    PROC PlotCirc(num Xcord,num Ycord,num Rad)
        IF ToolNum<>4 THEN
            Home;
            Plotter_Pickup;
        ELSE
            !Check position and move to safe position if needed
            !Check position and move to safe position if needed
            CurrentJoints:=CJointT();
            CurrentPos:=CalcRobT(CurrentJoints,tPlotter\WObj:=Bed1Wyong);

            IF (CurrentPos.trans.z<(Bed1Wyong.uframe.trans.z-30)) OR (((CurrentPos.trans.x+CurrentPos.extax.eax_a)>Bed1Wyong.uframe.trans.x) AND CurrentPos.trans.z<300) THEN
                !Robot in TS
                TPWrite("Jog robot out of tool station AND HOME");
                Stop;
            ENDIF
        ENDIF


        IF Rad<100 THEN
            vPlotter:=[10,5,2000,15];
        ELSE
            vPlotter:=[50,15,2000,15];
        ENDIF


        !Plot Circle
        Plotterc5.trans:=[(-1*Xcord),Ycord,PlotterZ];
        PlotterTemp.trans:=[Plotterc5.trans.x+Rad,Plotterc5.trans.y,PlotterZ];

        IF PlotterTemp.trans.y>0 THEN
            IF PlotterTemp.trans.y<(abs(tPlotter.tframe.trans.x)-10) THEN
                PlotterZOri:=ACos(PlotterTemp.trans.y/abs(tPlotter.tframe.trans.x));
                IF PlotterZOri>PlotA6Max THEN
                    PlotterZOri:=90;
                ENDIF
                PlotterTemp.rot:=OrientZYX(-90+PlotterZOri,0,180);
                PlotterTemp.trans.y:=PlotterTemp.trans.y-((abs(tPlotter.tframe.trans.x)-Ycord)*(9/((abs(tPlotter.tframe.trans.x)-540))));
            ELSEIF PlotterTemp.trans.y<2500 THEN
                PlotterZori:=25;
                PlotterTemp.rot:=OrientZYX(-90+PlotterZOri,0,180);
            ELSE
                PlotterTemp.rot:=OrientZYX(-90,0,180);
            ENDIF
        ELSE
            RAISE ERR_PLOT_POS;
        ENDIF

        IF PlotterTemp.trans.y+Bed1.uframe.trans.y>2800 THEN
            PlotterTemp.extax.eax_a:=(PlotterTemp.trans.x+Bed1Wyong.uframe.trans.x);
        ELSE
            PlotterTemp.extax.eax_a:=(PlotterTemp.trans.x+Bed1Wyong.uframe.trans.x+1000+Abs(tPlotter.tframe.trans.x*Sin(PlotterZOri)));
        ENDIF

        IF PlotterTemp.extax.eax_a>10150 THEN
            PlotterTemp.extax.eax_a:=10100;
        ELSEIF PlotterTemp.extax.eax_a<0 THEN
            PlotterTemp.extax.eax_a:=0;
        ENDIF

        WaitTime\inpos,0.1;
        ConfJ\Off;
        ConfL\Off;

        MoveJ Offs(PlotterTemp,0,0,50),v1500,z5,tPlotter\WObj:=Bed1Wyong;
        MoveL PlotterTemp,v10,fine,tPlotter\WObj:=Bed1Wyong;

        PlotterTemp2.trans:=[Plotterc5.trans.x,Plotterc5.trans.y+Rad,PlotterZ];
        IF PlotterTemp2.trans.y>0 THEN
            IF PlotterTemp2.trans.y<(abs(tPlotter.tframe.trans.x)-10) THEN
                PlotterZOri:=ACos(PlotterTemp2.trans.y/abs(tPlotter.tframe.trans.x));
                IF PlotterZOri>PlotA6Max THEN
                    PlotterZOri:=90;
                ENDIF
                PlotterTemp2.rot:=OrientZYX(-90+PlotterZOri,0,180);
                PlotterTemp2.trans.y:=PlotterTemp2.trans.y-((abs(tPlotter.tframe.trans.x)-(Ycord+Rad))*(9/((abs(tPlotter.tframe.trans.x)-540))));
            ELSEIF PlotterTemp2.trans.y<2500 THEN
                PlotterZori:=25;
                PlotterTemp2.rot:=OrientZYX(-90+PlotterZOri,0,180);
            ELSE
                PlotterZOri:=0;
                PlotterTemp2.rot:=OrientZYX(-90,0,180);
            ENDIF
        ELSE
            RAISE ERR_PLOT_POS;
        ENDIF
        IF PlotterTemp2.trans.y+Bed1.uframe.trans.y>2800 THEN
            PlotterTemp2.extax.eax_a:=(PlotterTemp2.trans.x+Bed1Wyong.uframe.trans.x);
        ELSE
            PlotterTemp2.extax.eax_a:=(PlotterTemp2.trans.x+Bed1Wyong.uframe.trans.x+1000+Abs(tPlotter.tframe.trans.x*Sin(PlotterZOri)));
        ENDIF

        IF PlotterTemp2.extax.eax_a>10150 THEN
            PlotterTemp2.extax.eax_a:=10100;
        ELSEIF PlotterTemp2.extax.eax_a<0 THEN
            PlotterTemp2.extax.eax_a:=0;
        ENDIF

        PlotterTemp3.trans:=[Plotterc5.trans.x-Rad,Plotterc5.trans.y,PlotterZ];
        IF PlotterTemp3.trans.y>0 THEN
            IF PlotterTemp3.trans.y<(abs(tPlotter.tframe.trans.x)-10) THEN
                PlotterZOri:=ACos(PlotterTemp3.trans.y/abs(tPlotter.tframe.trans.x));
                IF PlotterZOri>PlotA6Max THEN
                    PlotterZOri:=90;
                ENDIF
                PlotterTemp3.rot:=OrientZYX(-90+PlotterZOri,0,180);
                PlotterTemp3.trans.y:=PlotterTemp3.trans.y-((abs(tPlotter.tframe.trans.x)-(Ycord-Rad))*(9/((abs(tPlotter.tframe.trans.x)-540))));

            ELSEIF PlotterTemp3.trans.y<2500 THEN
                PlotterZori:=25;
                PlotterTemp3.rot:=OrientZYX(-90+PlotterZOri,0,180);
            ELSE
                PlotterZOri:=0;
                PlotterTemp3.rot:=OrientZYX(-90,0,180);
            ENDIF
        ELSE
            RAISE ERR_PLOT_POS;
        ENDIF
        IF PlotterTemp3.trans.y+Bed1Wyong.uframe.trans.y>2800 THEN
            PlotterTemp3.extax:=[(PlotterTemp3.trans.x+Bed1Wyong.uframe.trans.x),9E+09,9E+09,9E+09,9E+09,9E+09];
        ELSE
            PlotterTemp3.extax:=[(PlotterTemp3.trans.x+Bed1Wyong.uframe.trans.x+1000+Abs(tPlotter.tframe.trans.x*Sin(PlotterZOri))),9E+09,9E+09,9E+09,9E+09,9E+09];
        ENDIF

        IF PlotterTemp3.extax.eax_a>10150 THEN
            PlotterTemp3.extax.eax_a:=10100;
        ELSEIF PlotterTemp3.extax.eax_a<0 THEN
            PlotterTemp3.extax.eax_a:=0;
        ENDIF
        MoveC PlotterTemp2,PlotterTemp3,vPlotter,fine,tPlotter\WObj:=Bed1Wyong;

        PlotterTemp.trans:=[Plotterc5.trans.x,Plotterc5.trans.y-Rad,PlotterZ];
        IF PlotterTemp.trans.y>0 THEN
            IF PlotterTemp.trans.y<(abs(tPlotter.tframe.trans.x)-10) THEN
                PlotterZOri:=ACos(PlotterTemp.trans.y/abs(tPlotter.tframe.trans.x));
                IF PlotterZOri>PlotA6Max THEN
                    PlotterZOri:=90;
                ENDIF
                PlotterTemp.rot:=OrientZYX(-90+PlotterZOri,0,180);
                PlotterTemp.trans.y:=PlotterTemp.trans.y-((abs(tPlotter.tframe.trans.x)-(Ycord-Rad))*(9/((abs(tPlotter.tframe.trans.x)-540))));
            ELSE
                PlotterZOri:=0;
                PlotterTemp.rot:=OrientZYX(-90,0,180);
            ENDIF
        ELSE
            RAISE ERR_PLOT_POS;
        ENDIF

        IF PlotterTemp.trans.y+Bed1.uframe.trans.y>2800 THEN
            PlotterTemp.extax:=[(PlotterTemp.trans.x+Bed1Wyong.uframe.trans.x),9E+09,9E+09,9E+09,9E+09,9E+09];
        ELSE
            PlotterTemp.extax:=[(PlotterTemp.trans.x+Bed1Wyong.uframe.trans.x+1000+Abs(tPlotter.tframe.trans.x*Sin(PlotterZOri))),9E+09,9E+09,9E+09,9E+09,9E+09];
        ENDIF

        IF PlotterTemp.extax.eax_a>10150 THEN
            PlotterTemp.extax.eax_a:=10100;
        ELSEIF PlotterTemp.extax.eax_a<0 THEN
            PlotterTemp.extax.eax_a:=0;
        ENDIF

        PlotterTemp2.trans:=[Plotterc5.trans.x+Rad,Plotterc5.trans.y,PlotterZ];
        IF PlotterTemp2.trans.y>0 THEN
            IF PlotterTemp2.trans.y<(abs(tPlotter.tframe.trans.x)-10) THEN
                PlotterZOri:=ACos(PlotterTemp2.trans.y/abs(tPlotter.tframe.trans.x));
                IF PlotterZOri>PlotA6Max THEN
                    PlotterZOri:=90;
                ENDIF
                PlotterTemp2.rot:=OrientZYX(-90+PlotterZOri,0,180);
                PlotterTemp2.trans.y:=PlotterTemp2.trans.y-((abs(tPlotter.tframe.trans.x)-(Ycord))*(9/((abs(tPlotter.tframe.trans.x)-540))));
            ELSE
                PlotterZOri:=0;
                PlotterTemp2.rot:=OrientZYX(-90,0,180);
            ENDIF
        ELSE
            RAISE ERR_PLOT_POS;
        ENDIF
        IF PlotterTemp2.trans.y+Bed1.uframe.trans.y>2800 THEN
            PlotterTemp2.extax.eax_a:=(PlotterTemp2.trans.x+Bed1Wyong.uframe.trans.x);
        ELSE
            PlotterTemp2.extax.eax_a:=(PlotterTemp2.trans.x+Bed1Wyong.uframe.trans.x+1000+Abs(tPlotter.tframe.trans.x*Sin(PlotterZOri)));
        ENDIF

        IF PlotterTemp2.extax.eax_a>10150 THEN
            PlotterTemp2.extax.eax_a:=10100;
        ELSEIF PlotterTemp2.extax.eax_a<0 THEN
            PlotterTemp2.extax.eax_a:=0;
        ENDIF
        MoveC PlotterTemp,PlotterTemp2,vPlotter,fine,tPlotter\WObj:=Bed1Wyong;
        MoveL Offs(PlotterTemp2,0,0,50),v100,z5,tPlotter\WObj:=Bed1Wyong;
        MoveJ Offs(PlotterTemp2,0,0,200),v500,fine,tPlotter\WObj:=Bed1Wyong;
        ConfJ\On;
        ConfL\On;

    ERROR
        RAISE ;

    ENDPROC

    PROC PackAway()
        !VAR jointtarget jtTarget;
        Home;
        !jtTarget := [[138.31,-55.47,60.29,-0.02,84.30,-2.02], [9416.99,9E+09,9E+09,9E+09,9E+09,9E+09]];
        !MoveAbsJ jtTarget, v500, fine, tTCMaster;
        MoveJ pHomeLoadout,v500,z50,tTCMaster;
    ERROR
        RAISE ;
    ENDPROC


    PROC Home()
        !Move robot to safe position, drop off any tools, close tool boxes

        TEST ToolNum

        CASE 1:
            !TCmaster
            !Check for any tb lids open and robot in tool stations
            !Move to Home
            CurrentJoints:=CJointT();
            CurrentPos:=CalcRobT(CurrentJoints,tTCMaster\WObj:=wobj0);

            IF (CurrentPos.trans.x)>8000 AND (CurrentPos.trans.z<265) THEN
                TPErase;
                TPWrite("Jog robot out of tool station AND HOME");
                Stop;
            ENDIF

        CASE 2:
            !Heli
            CurrentJoints:=CJointT();
            CurrentPos:=CalcRobT(CurrentJoints,tHeli\WObj:=wobj0);

            IF (CurrentPos.trans.x)>8000 AND CurrentPos.trans.z<125 THEN
                TPWrite("Jog robot out of tool station AND HOME");
                Stop;
            ENDIF

            IF CurrentPos.trans.y>(Bed1.uframe.trans.y+3000) THEN
                MoveL Offs(CurrentPos,0,(3000-CurrentPos.trans.y),50),v10,z5,tHeli\WObj:=wobj0;
                MoveJ Offs(CurrentPos,0,(3000-CurrentPos.trans.y),300-CurrentPos.trans.z),v100,z5,tHeli\WObj:=wobj0;
            ENDIF
            Heli_Dropoff;

        CASE 3:
            !VS

            CurrentJoints:=CJointT();
            CurrentPos:=CalcRobT(CurrentJoints,tVS\WObj:=wobj0);


            IF (CurrentPos.trans.x)>8000 AND CurrentPos.trans.z<265 THEN
                TPErase;
                TPWrite("Jog robot out of tool station AND HOME");
                Stop;
            ELSEIF CurrentPos.trans.z<200 THEN
                MoveL Offs(CurrentPos,0,0,(200-CurrentPos.trans.z)),v500,z5,tVS;

            ENDIF


            VS_Dropoff;


        CASE 4:
            !Plotter

            CurrentJoints:=CJointT();
            CurrentPos:=CalcRobT(CurrentJoints,tPlotter\WObj:=wobj0);

            IF CurrentPos.trans.z<270 AND (CurrentPos.trans.x)<8000 THEN
                MoveL Offs(CurrentPos,0,0,(270-CurrentPos.trans.z)),v500,z5,tPlotter;
            ENDIF

            IF (CurrentPos.trans.x)>8000 AND CurrentPos.trans.z<265 THEN
                TPErase;
                TPWrite("Jog robot out of tool station AND HOME");
                Stop;
            ENDIF

            IF CurrentPos.trans.y>(Bed1.uframe.trans.y+3300) THEN
                MoveL Offs(CurrentPos,0,(3300-CurrentPos.trans.y),50),v10,z5,tPlotter\WObj:=wobj0;
                MoveJ Offs(CurrentPos,0,(3300-CurrentPos.trans.y),1000-CurrentPos.trans.z),v100,z5,tPlotter\WObj:=wobj0;
            ENDIF
            Plotter_Dropoff;

        CASE 5:
            CurrentJoints:=CJointT();
            CurrentPos:=CalcRobT(CurrentJoints,tVac\WObj:=wobj0);

            IF (CurrentPos.trans.x)>8000 AND CurrentPos.trans.z<265 THEN
                TPErase;
                TPWrite("Jog robot out of tool station AND HOME");
                Stop;
            ENDIF
            IF CurrentPos.trans.z<200 AND (CurrentPos.trans.x)<8000 THEN
                MoveL Offs(CurrentPos,0,0,(200-CurrentPos.trans.z)),v500,fine,tVac;
            ENDIF
            CurrentJoints:=CJointT();
            CurrentPos:=CalcRobT(CurrentJoints,tVac\WObj:=wobj0);
            IF CurrentPos.trans.y>(Bed1.uframe.trans.y+3000) THEN
                MoveL Offs(CurrentPos,0,(3000-CurrentPos.trans.y),50),v200,z5,tVac\WObj:=wobj0;
                MoveJ Offs(CurrentPos,0,(3000-CurrentPos.trans.y),700-CurrentPos.trans.z),v200,z5,tVac\WObj:=wobj0;
            ENDIF
            Vac_Dropoff;

        CASE 6:
            CurrentJoints:=CJointT();
            CurrentPos:=CalcRobT(CurrentJoints,tPolish\WObj:=wobj0);


            IF (CurrentPos.trans.x)>8000 AND CurrentPos.trans.z<265 THEN
                TPErase;
                TPWrite("Jog robot out of tool station AND HOME");
                Stop;

            ENDIF
            Polish_Dropoff;

        DEFAULT:
            !Unknown
            RAISE ERR_TC_SELECTION;

        ENDTEST

        MoveJ pHome,v500,fine,tTCMaster;

    ERROR
        RAISE ;

    ENDPROC

    FUNC num PointToPointDist(num px,num py,num x1,num y1)
        !Used to check if point is within helicopter blades

        VAR num Dist;

        Dist:=Sqrt((x1-px)*(x1-px)+(y1-py)*(y1-py));
        RETURN Dist;
    ENDFUNC

    FUNC num HighestArray(num count)
        !Used to determine highest height offset
        VAR num j;
        VAR num HighestValue;
        HighestValue:=HeliZArray{1};
        FOR j FROM 1 TO count DO
            IF HeliZArray{j}>HighestValue THEN
                HighestValue:=HeliZArray{j};
            ENDIF
        ENDFOR
        IF PreviousHighest>HighestValue THEN
            PreviousHighest:=HighestValue;
            RETURN PreviousHighest;
        ELSEIF HighestValue<=-30 THEN
            PreviousHighest:=HighestValue;
            RETURN 0;
        ELSE
            PreviousHighest:=HighestValue;
            RETURN HighestValue;
        ENDIF

    ENDFUNC

    PROC HeliZ(num x1,num y1,bool ResetZArray)
        !Determines height offsets for helicopter movements
        VAR num CloseYPos;
        x1:=Abs(x1);
        IF ResetZArray=TRUE THEN
            HeliZArrayCounter:=1;
            FOR i FROM 1 TO DIM(HeliZArray,1) DO
                HeliZArray{i}:=-50;
            ENDFOR
        ENDIF

        FOR i FROM 1 TO 17 DO
            FOR j FROM 1 TO 4 DO
                IF PointToPointDist(x1,y1,BedZpos{j,i,1},BedZpos{j,i,2})<=HeliBladeWidth/2 THEN
                    HeliZArray{HeliZArrayCounter}:=BedZreads{j,i};
                    Incr HeliZArrayCounter;
                ENDIF
            ENDFOR
        ENDFOR

    ENDPROC

    PROC PlotBedGrid(num Xcord1,num Ycord1,num ZOffset)
        !Used by BedGridPlotter for Z datum
        Plotterp1.trans:=[Xcord1,Ycord1,200+ZOffset];
        !+46

        IF Plotterp1.trans.y>0 THEN
            IF Plotterp1.trans.y<(abs(tPlotter.tframe.trans.x)-10) THEN
                PlotterZOri:=ACos(Plotterp1.trans.y/abs(tPlotter.tframe.trans.x));
                IF PlotterZOri>PlotA6Max THEN
                    PlotterZOri:=90;
                ENDIF
                Plotterp1.rot:=OrientZYX(-90+PlotterZOri,0,180);
            ELSE
                PlotterZOri:=0;
                Plotterp1.rot:=OrientZYX(-90,0,180);
            ENDIF
        ELSE
            RAISE ERR_PLOT_POS;
        ENDIF

        IF PlotterP1.trans.y>(abs(tPlotter.tframe.trans.x)+250) THEN
            Plotterp1.extax:=[(Plotterp1.trans.x+Bed1.uframe.trans.x),9E+09,9E+09,9E+09,9E+09,9E+09];
        ELSE
            Plotterp1.extax:=[(Plotterp1.trans.x+Bed1.uframe.trans.x+1000+Abs(tPlotter.tframe.trans.x*Sin(PlotterZOri))),9E+09,9E+09,9E+09,9E+09,9E+09];
        ENDIF

        IF Plotterp1.extax.eax_a>10150 THEN
            Plotterp1.extax.eax_a:=10100;
        ENDIF

        IF Plotterp1.extax.eax_a<0 THEN
            Plotterp1.extax.eax_a:=0;
        ENDIF

        vPlotter:=[100,15,2000,15];

        MoveL Plotterp1,v300,zPlotter,tTCMaster\WObj:=Bed1Wyong;

    ENDPROC

    PROC BedGridPlotter()
        !Get Z datum offset
        FOR k FROM 7 TO 19 DO
            !Move x
            FOR j FROM 4 TO 9 DO
                !Move y

                PlotBedGrid(k*XGridSpacing+100),(j*YGridSpacing+100),Bed1Zread{10-j,(k+1)};
                WaitTime\inpos,0.1;

            ENDFOR

        ENDFOR

    ENDPROC

    PROC MoveGridDatum()
        !Sweep across bed maintaining Z height through offsets
        FOR j FROM 9 TO 4 DO
            FOR k FROM 11 TO 1 DO
                !Move x
                PlotBedGrid(k*XGridSpacing+100),(j*YGridSpacing+100),Bed1Zread{10-j,(k+1)};
            ENDFOR
        ENDFOR
    ENDPROC


    PROC VacuumBed()

        VAR num VacOverlap:=-400;
        IF ToolNum<>5 THEN
            Home;
            Vac_Pickup;
        ELSE
            CurrentJoints:=CJointT();
            CurrentPos:=CalcRobT(CurrentJoints,tVac\WObj:=Bed1Wyong);
            IF CurrentPos.trans.x<0 AND (CurrentPos.trans.z<150) THEN
                MoveL Offs(CurrentPos,0,0,(150-CurrentPos.trans.z)),v500,z5,tVac\WObj:=Bed1Wyong;
            ELSEIF (CurrentPos.trans.z<700) THEN
                MoveL Offs(CurrentPos,0,0,(700-CurrentPos.trans.z)),v500,z5,tVac\WObj:=Bed1Wyong;
            ENDIF
        ENDIF

        pTemp:=pVacStart;
        pTemp2:=pVacStart;
        pTemp2.trans.x:=pVacStart2.trans.x;
        pTemp2.extax.eax_a:=pVacStart2.extax.eax_a;

        Vac_on;
        FOR i FROM 0 TO (Round((pVacStart.trans.y-pVacStart2.trans.y)/(-1*VacOverlap))) DO
            IF pTemp.trans.y+i*VacOverlap>pVacStart2.trans.y THEN
                MoveJ Offs(pTemp,0,i*VacOverlap,150),v500,z5,tVac\WObj:=Bed1Wyong;
                MoveL Offs(pTemp,0,i*VacOverlap,0),v50,z5,tVac\WObj:=Bed1Wyong;
                MoveL Offs(pTemp2,0,i*VacOverlap,0),v100,z5,tVac\WObj:=Bed1Wyong;
                MoveL Offs(pTemp2,0,i*VacOverlap,150),v50,fine,tVac\WObj:=Bed1Wyong;
            ENDIF
        ENDFOR

        Vac_off;

        CurrentJoints:=CJointT();
        CurrentPos:=CalcRobT(CurrentJoints,tVac\WObj:=wobj0);
        MoveL Offs(CurrentPos,0,0,800-CurrentPos.trans.z),v100,z5,tVac\WObj:=wobj0;

    ENDPROC

    PROC JointPositions()

        VAR num PolishOverlap:=450;
        pPolTemp:=pPolStart1;
        pPolTemp2:=pPolStart1;
        pPolTemp2.extax.eax_a:=pPolStart1.extax.eax_a-7500;
        pPolTemp2.trans.x:=-7500;

        pPolTemp.rot:=pPolStart1.rot;
        pPolTemp2.rot:=pPolStart1.rot;

        pPolTemp2.rot:=pPolStart2.rot;
        pPolTemp2.extax.eax_a:=pPolStart1.extax.eax_a-8500;
        CurrentJoints5:=CJointT();
        CurrentJoints6:=CalcJointT(Offs(pPolTemp2,50,(1+1)*PolishOverlap,40),tPolish\WObj:=Bed1Wyong);

    ENDPROC


    PROC RobbiePlot()

        ! !Write R
        !PlotLine 6900,1000, 6900,2000;
        !PlotArc 6900,2000,6650,1750,6900,1500;
        !PlotLine 6900,1500,6650,1000;

        !!Write O
        !PlotArc 6300,2000, 6050,1500,6300,1000;
        !PlotArc 6300,1000, 6550,1500,6300,2000;

        !!Write B
        !PlotLine 5700,1000, 5700,2000;
        !PlotArc 5700,2000,5450,1750,5700,1500;
        !PlotArc 5700,1500,5450,1250,5700,1000;

        !!Write B
        !PlotLine 5100,1000, 5100,2000;
        !PlotArc 5100,2000,4850,1750,5100,1500;
        !PlotArc 5100,1500,4850,1250,5100,1000;

        !!Write I
        !PlotLine 4500,1000, 4500,2000;

        !!Write E
        !PlotLine 3900,1000, 3900,2000;
        !PlotLine 3900,2000, 3400,2000;
        !PlotLine 3900,1500, 3400,1500;
        !PlotLine 3900,1000, 3400,1000;

        !formbox
        PlotRect 2000,500,2000,3500,6000,3500,6000,500;
        !Ferrule
        WaitTime\inpos,0.1;
        PlotCirc 2250,750,(PlotCircleD/2);
        PlotLine(2250-PlotCircleD/2-CrossHairExt),750,(2250+PlotCircleD/2+CrossHairExt),750;
        PlotLine 2250,(750-PlotCircleD/2-CrossHairExt),2250,(750+PlotCircleD/2+CrossHairExt);
        !Ferrule
        WaitTime\inpos,0.1;
        PlotCirc 2250,3250,(PlotCircleD/2);
        PlotLine(2250-PlotCircleD/2-CrossHairExt),3250,(2250+PlotCircleD/2+CrossHairExt),3250;
        PlotLine 2250,(3250-PlotCircleD/2-CrossHairExt),2250,(3250+PlotCircleD/2+CrossHairExt);
        !Grout tube Casee 4
        WaitTime\inpos,0.1;
        iCoord1x:=6000;
        iCoord1y:=2000;
        iAngle:=0;
        PlotRect iCoord1x-GroutWidth/2*Sin(iAngle)-GroutHeight*Cos(iAngle),iCoord1y+GroutHeight*Sin(iAngle)-GroutWidth/2*Cos(iAngle),iCoord1x+GroutWidth/2*Sin(iAngle)-GroutHeight*Cos(iAngle),iCoord1y+GroutHeight*Sin(iAngle)+GroutWidth/2*Cos(iAngle),iCoord1x+GroutWidth/2*Sin(iAngle),iCoord1y+GroutWidth/2*Cos(iAngle),iCoord1x-GroutWidth/2*Sin(iAngle),iCoord1y-GroutWidth/2*Cos(iAngle);

        !Lifting points 180 angle
        WaitTime\inpos,0.1;
        TriangleAngle:=180;
        iCoord1x:=5000;
        iCoord1y:=3500;
        PlotLine iCoord1x-TriangleHeight*Sin(TriangleAngle),iCoord1y-TriangleHeight*Cos(TriangleAngle),iCoord1x-TriangleBase/2*Cos(TriangleAngle),iCoord1y+TriangleBase/2*Sin(TriangleAngle);
        PlotLine iCoord1x-TriangleBase/2*Cos(TriangleAngle),iCoord1y+TriangleBase/2*Sin(TriangleAngle),iCoord1x+TriangleBase/2*Cos(TriangleAngle),iCoord1y-TriangleBase/2*Sin(TriangleAngle);
        PlotLine iCoord1x+TriangleBase/2*Cos(TriangleAngle),iCoord1y-TriangleBase/2*Sin(TriangleAngle),iCoord1x-TriangleHeight*Sin(TriangleAngle),iCoord1y-TriangleHeight*Cos(TriangleAngle);
        !Lifting points 180 angle
        WaitTime\inpos,0.1;
        TriangleAngle:=180;
        iCoord1x:=3000;
        iCoord1y:=3500;
        PlotLine iCoord1x-TriangleHeight*Sin(TriangleAngle),iCoord1y-TriangleHeight*Cos(TriangleAngle),iCoord1x-TriangleBase/2*Cos(TriangleAngle),iCoord1y+TriangleBase/2*Sin(TriangleAngle);
        PlotLine iCoord1x-TriangleBase/2*Cos(TriangleAngle),iCoord1y+TriangleBase/2*Sin(TriangleAngle),iCoord1x+TriangleBase/2*Cos(TriangleAngle),iCoord1y-TriangleBase/2*Sin(TriangleAngle);
        PlotLine iCoord1x+TriangleBase/2*Cos(TriangleAngle),iCoord1y-TriangleBase/2*Sin(TriangleAngle),iCoord1x-TriangleHeight*Sin(TriangleAngle),iCoord1y-TriangleHeight*Cos(TriangleAngle);

        Plotter_Dropoff;

    ENDPROC

    PROC PolishDemo()
        IF ToolNum<>6 THEN
            Home;
            Polish_Pickup;
        ELSE
            CurrentJoints:=CJointT();
            CurrentPos:=CalcRobT(CurrentJoints,tPolish\WObj:=wobj0);
            IF CurrentPos.trans.z<600 THEN
                MoveL Offs(CurrentPos,0,0,(600-CurrentPos.trans.z)),v500,z5,tPolish;
            ENDIF
        ENDIF
        MoveJ pPolHome,v500,z5,tPolish;
        pPolTemp:=pPolStart1;
        pPolTemp2:=pPolStart1;
        pPolTemp2.extax.eax_a:=pPolStart1.extax.eax_a-7500;
        pPolTemp2.trans.x:=-7500;
        pPolTemp.rot:=pPolStart1.rot;
        pPolTemp2.rot:=pPolStart1.rot;
        FCCalib PolishLoad;
        pPolTemp.extax.eax_a:=pPolStart1.extax.eax_a;
        MoveJ Offs(pPolTemp,0,0,100),v500,z5,tPolish\WObj:=Bed1Wyong;
        Pol_on;
        MoveL Offs(pPolTemp,0,0,50),v100,fine,tPolish\WObj:=Bed1Wyong;
        myForceVector:=FCGetForce(\Tool:=tPolish);
        FCPress1LStart Offs(pPolTemp,-25,0,55),v10,\Fz:=120,15,\ForceChange:=50\PosSupvDist:=125,z5,tPolish\WObj:=Bed1Wyong;
        pPolTemp2.extax.eax_a:=pPolStart2.extax.eax_a-300;
        FCPressL Offs(pPolTemp2,-300,0,-15),v100,130,fine,tPolish\WObj:=Bed1Wyong;
        FCPressEnd Offs(pPolTemp2,-300,0,75),v50,\DeactOnly,tPolish\WObj:=Bed1Wyong;
        CurrentJoints:=CJointT();
        CurrentPos:=CalcRobT(CurrentJoints,tPolish\WObj:=Bed1Wyong);
        MoveJ Offs(Reltool(CurrentPos,0,0,-100),0,450,0),v100,fine,tPolish\WObj:=Bed1Wyong;
        Pol_off;
        Polish_Dropoff;
    ENDPROC



    PROC BedGrid()

        !        MoveJ Offs(p10Maps,500*(1-1)+2000*(1-1),650*(1-1),50),v500,z5,tTCMaster\WObj:=Bed1Wyong;
        !        MoveL Offs(p10Maps,500*(1-1)+2000*(1-1),650*(1-1),0),v500,fine,tTCMaster\WObj:=Bed1Wyong;
        !        Stop;
        !        MoveL Offs(p10Maps,500*(1-1)+2000*(1-1),650*(1-1),50),v500,z5,tTCMaster\WObj:=Bed1Wyong;
        !        Stop;

        FOR i FROM 1 TO 5 DO
            !Move EAX
            FOR k FROM 1 TO 4 DO
                !Move x
                FOR j FROM 1 TO 4 DO
                    !Move y
                    IF 500*(k-1)+2000*(i-1)<8001 THEN
                        p10maps.extax.eax_a:=Bed1Wyong.uframe.trans.x+p10Maps.trans.x-500*(k-1)-2000*(i-1);
                        IF p10maps.extax.eax_a>10150 THEN
                            p10maps.extax.eax_a:=10100;
                        ENDIF
                        IF p10maps.extax.eax_a<1000 THEN
                            p10maps.extax.eax_a:=1000;
                        ENDIF

                        !MoveJ Offs(p10Maps,-500*(k-1)-2000*(i-1),650*(j-1),50),v500,z5,tTCMaster\WObj:=Bed1Wyong;
                        !MoveL Offs(p10Maps,-500*(k-1)-2000*(i-1),650*(j-1),0),v500,fine,tTCMaster\WObj:=Bed1Wyong;
                        !TPReadNum BedZread,"Enter Z reading";
                        !BedZreads{5-j,((i-1)*4+k)}:=BedZread;
                        BedZpos{5-j,((i-1)*4+k),1}:=p10Maps.trans.x-500*(k-1)-2000*(i-1);
                        BedZpos{5-j,((i-1)*4+k),2}:=p10maps.trans.y+650*(j-1);
                        !MoveL Offs(p10Maps,-500*(k-1)-2000*(i-1),650*(j-1),50),v500,z5,tTCMaster\WObj:=Bed1Wyong;
                    ENDIF

                ENDFOR
            ENDFOR
        ENDFOR
        Stop;

    ENDPROC


    PROC ClearBedZ()

        FOR i FROM 1 TO 4 DO
            !Move EAX
            FOR k FROM 1 TO 24 DO
                !Move x
                BedZreads{i,k}:=0;
                BedZpos{i,k,1}:=0;
                BedZpos{i,k,2}:=0;
            ENDFOR
        ENDFOR

    ENDPROC




    PROC BHTestTask()
        TPErase;
        TPWrite "BH Test Task";
        TPWrite "Press Play to confirm and start task";
        Stop;

        TPErase;
        TPWrite "Starting BH Test Task...";

        Heli_Pickup;
        MoveJ Offs(ptHeli,0,0,1000),v500,fine,tHeli;
        TPWrite "Helicopter tool at 1000mm above pickup";
        WaitTime 2;

        Heli_Dropoff;
        TPWrite "Helicopter tool dropped off";

        Polish_Pickup;
        MoveJ Offs(ptPolish,0,0,1000),v500,fine,tPolish;
        TPWrite "Polisher tool at 1000mm above pickup";
        WaitTime 2;

        Polish_Dropoff;
        TPWrite "Polisher tool dropped off";

        Home;
        TPWrite "BH Test Task Complete";

    ERROR
        RAISE ;
    ENDPROC



    PROC Datum()
        ! Datum - draws small circle at Bed1Wyong origin (0,0)
        ! Generated by Onyx Toolpath Generator
        VAR robtarget pDatumCenter;
        VAR robtarget pDatumCircle;
        VAR num DatumZ:=0;
        VAR num DatumRadius:=100;
        VAR num SafeZ:=500;
        VAR num i;

        TPWrite "Datum: ToolNum=" \Num:=ToolNum;
        IF ToolNum<>4 THEN
            TPWrite "No plotter! Will pickup plotter.";
            Stop;
            Home;
            Plotter_Pickup;
        ELSE
            CurrentJoints:=CJointT();
            CurrentPos:=CalcRobT(CurrentJoints,tPlotter\WObj:=wobj0);
            IF CurrentPos.trans.z<600 THEN
                MoveL Offs(CurrentPos,0,0,(600-CurrentPos.trans.z)),v500,z5,tPlotter;
            ENDIF
        ENDIF

        ConfL\Off;
        ConfJ\Off;

        pDatumCenter:=[[0,0,DatumZ],[0,0,1,0],[0,0,0,0],[0,9E+09,9E+09,9E+09,9E+09,9E+09]];
        pDatumCenter.rot:=OrientZYX(-90,0,180);
        pDatumCenter.extax.eax_a:=6500;

        TPWrite "Datum: Drawing circle at origin";
        TPWrite "Press Play to continue";
        Stop;

        pDatumCircle:=pDatumCenter;
        pDatumCircle.trans.z:=SafeZ;
        MoveJ pDatumCircle,v500,z5,tPlotter\WObj:=Bed1Wyong;

        pDatumCircle.trans.x:=DatumRadius;
        pDatumCircle.trans.z:=DatumZ;
        MoveJ pDatumCircle,v500,z5,tPlotter\WObj:=Bed1Wyong;

        FOR i FROM 1 TO 8 DO
            pDatumCircle.trans.x:=DatumRadius*Cos(i*45);
            pDatumCircle.trans.y:=DatumRadius*Sin(i*45);
            MoveJ pDatumCircle,v100,fine,tPlotter\WObj:=Bed1Wyong;
        ENDFOR

        pDatumCircle.trans.x:=0;
        pDatumCircle.trans.y:=0;
        pDatumCircle.trans.z:=DatumZ;
        MoveJ pDatumCircle,v100,fine,tPlotter\WObj:=Bed1Wyong;

        TPWrite "Plotter at datum center (0,0)";
        TPWrite "Press Play to return tool";
        Stop;

        pDatumCircle.trans.z:=SafeZ;
        MoveJ pDatumCircle,v500,z5,tPlotter\WObj:=Bed1Wyong;

        ConfL\On;
        ConfJ\On;

        Plotter_Dropoff;
        Home;

        TPWrite "Datum Complete";
    ERROR
        RAISE;
    ENDPROC


    PROC PyHeli()
        ! PyHeli - Helicopter serpentine pattern
        ! Workzone: panel
        ! Force Control ENABLED: 300N (ramping 10%->100% over 5s)
        ! Generated by Onyx Toolpath Generator

        VAR robtarget pHeliPos;
        VAR robtarget pHeliEnd;
        VAR num HeliZ:=150;
        VAR num SafeZ:=500;

        ! Workspace bounds (with offsets applied)
        VAR num WorkMinX:=1900;
        VAR num WorkMaxX:=6550;
        VAR num WorkMinY:=700;
        VAR num WorkMaxY:=2100;

        ! Pattern parameters
        VAR num StepSize:=450;
        VAR num SweepDir:=1;
        VAR num StepDir:=-1;
        VAR num CurrentY:=2100;
        VAR num CurrentX:=1900;
        VAR num NextY;
        VAR num NextX;
        VAR num StartX;
        VAR num EndX;
        VAR num StartY;
        VAR num EndY;

        ! Speed and blade parameters
        VAR num HeliSpeed:=100;
        VAR num HeliAngle:=8;
        VAR speeddata vHeliTravel:=[500,15,2000,15];
        VAR num NumPasses;
        VAR num HeliForce:=300;
        VAR num CurrentForce:=300;
        VAR clock RampClock;
        VAR bool bRamping:=FALSE;

        NumPasses:=Trunc(Abs(WorkMaxY-WorkMinY)/StepSize)+1;

        TPWrite "PyHeli: Serpentine Pattern";
        TPWrite "Work Area (6550,2100) to (1900,700)";
        TPWrite "Passes=" \Num:=NumPasses;
        TPWrite "Step=" \Num:=StepSize;
        TPWrite "Force=ON 300N";

        IF ToolNum<>2 THEN
            TPWrite "PyHeli: ToolNum<>2, need pickup";
            Stop;
            Home;
            Heli_Pickup;
        ELSE
            CurrentJoints:=CJointT();
            CurrentPos:=CalcRobT(CurrentJoints,tHeli\WObj:=Bed1Wyong);
            IF CurrentPos.trans.z<SafeZ THEN
                MoveL Offs(CurrentPos,0,0,(SafeZ-CurrentPos.trans.z)),v500,z5,tHeli\WObj:=Bed1Wyong;
            ENDIF
        ENDIF

        ! Set start/end based on sweep direction
        IF SweepDir=1 THEN
            StartX:=WorkMinX;
            EndX:=WorkMaxX;
        ELSE
            StartX:=WorkMaxX;
            EndX:=WorkMinX;
        ENDIF

        ! Set initial position with fixed orientation
        pHeliPos:=[[0,0,HeliZ],OrientZYX(0,0,180),[0,0,0,0],[0,9E+09,9E+09,9E+09,9E+09,9E+09]];

        ! Move to row start above surface (HOVER)
        pHeliPos.trans.x:=-StartX;
        pHeliPos.trans.y:=CurrentY;
        pHeliPos.trans.z:=SafeZ;
        pHeliPos.extax.eax_a:=Bed1Wyong.uframe.trans.x-StartX;
        MoveJ pHeliPos,v500,z5,tHeli\WObj:=Bed1Wyong;

        ! Disable configuration tracking for serpentine movements
        ConfL\Off;
        ConfJ\Off;

        ! Home stepper before setting blade angle (ensures StepperPos is valid)
        TPWrite "Homing blade stepper...";
        Heli_Stepper_Home;
        TPWrite "Stepper homed";

        ! Set blade angle while hovering
        TPWrite "Setting blade angle to " \Num:=HeliAngle;
        HeliBlade_Angle HeliAngle;
        WaitTime 2;
        TPWrite "Blade angle set";

        ! Calibrate force sensor while stationary (before blade spin)
        TPWrite "Calibrating force sensor...";
        FCCalib HeliLoad140rpm;
        TPWrite "Force sensor calibrated";

        TPWrite "Hovering over workspace - Press Play to start";
        Stop;

        ! Start blade rotation BEFORE lowering
        TPWrite "Starting blade rotation...";
        HeliBladeSpeed HeliSpeed,"FWD";
        WaitTime 1;

        ! Lower to working height
        TPWrite "Lowering to work surface...";
        pHeliPos.trans.z:=HeliZ;
        MoveL pHeliPos,v50,fine,tHeli\WObj:=Bed1Wyong;

        ! Start force control at 10% of target
        CurrentForce:=HeliForce*0.1;
        FCPress1LStart Offs(pHeliPos,0,0,25),v50,\Fz:=CurrentForce,15,\ForceChange:=50\PosSupvDist:=100,z5,tHeli\WObj:=Bed1Wyong;

        ! Start ramp timer - will ramp to 100% over 5 seconds during first sweep
        ClkReset RampClock;
        ClkStart RampClock;
        bRamping:=TRUE;
        TPWrite "Force ramping: 10% -> 100% over 5s";

        ! Set up end position for first sweep
        pHeliEnd:=pHeliPos;
        pHeliEnd.trans.x:=-EndX;
        pHeliEnd.extax.eax_a:=Bed1Wyong.uframe.trans.x-EndX;

        ! ========== PASS 1: X-direction sweeps (stepping in Y) ===========
        WHILE TRUE DO
            ! === SWEEP X (full length) ===
            FCPressL pHeliEnd,vHeliTravel,CurrentForce,fine,tHeli\WObj:=Bed1Wyong;

            ! Update force ramp if still ramping (applied on next move)
            IF bRamping THEN
                IF ClkRead(RampClock)>=5 THEN
                    CurrentForce:=HeliForce;
                    bRamping:=FALSE;
                    TPWrite "Force ramp complete: " \Num:=CurrentForce;
                ELSE
                    CurrentForce:=HeliForce*(0.1+0.9*ClkRead(RampClock)/5);
                ENDIF
            ENDIF

            ! Calculate next row
            NextY:=CurrentY+(StepDir*StepSize);

            ! Check if pass complete
            IF (StepDir=1 AND NextY>WorkMaxY) OR (StepDir=-1 AND NextY<WorkMinY) THEN
                EXIT;
            ENDIF

            ! Clamp to bounds
            IF NextY>WorkMaxY THEN
                NextY:=WorkMaxY;
            ELSEIF NextY<WorkMinY THEN
                NextY:=WorkMinY;
            ENDIF

            ! Step to next Y row
            pHeliEnd.trans.y:=NextY;
            FCPressL pHeliEnd,vHeliTravel,CurrentForce,fine,tHeli\WObj:=Bed1Wyong;
            CurrentY:=NextY;

            ! Flip sweep direction
            SweepDir:=-SweepDir;
            IF SweepDir=1 THEN
                StartX:=WorkMinX;
                EndX:=WorkMaxX;
            ELSE
                StartX:=WorkMaxX;
                EndX:=WorkMinX;
            ENDIF

            ! Set up end position for next sweep
            pHeliEnd.trans.x:=-EndX;
            pHeliEnd.extax.eax_a:=Bed1Wyong.uframe.trans.x-EndX;
        ENDWHILE

        ! ========== PASS 2: Y-direction sweeps (stepping in X) ==========
        TPWrite "=== PASS 2 START ===";

        ! Reset for Y-direction passes - start from current position
        CurrentX:=Abs(pHeliEnd.trans.x);
        TPWrite "Pass2: CurrentX=" \Num:=CurrentX;
        TPWrite "Pass2: CurrentY=" \Num:=CurrentY;
        TPWrite "Pass2: WorkMinX=" \Num:=WorkMinX;
        TPWrite "Pass2: WorkMaxX=" \Num:=WorkMaxX;

        ! Determine step direction based on where Pass 1 ended
        ! At high X, step toward low X; at low X, step toward high X
        IF CurrentX>((WorkMinX+WorkMaxX)/2) THEN
            StepDir:=-1;
            TPWrite "Pass2: StepDir=-1 (toward MinX)";
        ELSE
            StepDir:=1;
            TPWrite "Pass2: StepDir=+1 (toward MaxX)";
        ENDIF

        ! Determine sweep direction based on where Pass 1 ended (which Y edge)
        IF CurrentY>((WorkMinY+WorkMaxY)/2) THEN
            SweepDir:=1;
            StartY:=WorkMaxY;
            EndY:=WorkMinY;
            TPWrite "Pass2: Sweep MinY first";
        ELSE
            SweepDir:=-1;
            StartY:=WorkMinY;
            EndY:=WorkMaxY;
            TPWrite "Pass2: Sweep MaxY first";
        ENDIF

        TPWrite "Pass2: EndY=" \Num:=EndY;

        ! First Y sweep from current position
        TPWrite "Pass2: First Y sweep...";
        pHeliEnd.trans.y:=EndY;
        FCPressL pHeliEnd,vHeliTravel,CurrentForce,fine,tHeli\WObj:=Bed1Wyong;
        TPWrite "Pass2: First Y sweep done";

        TPWrite "Pass2: Entering X-step loop";

        WHILE TRUE DO
            ! Calculate next column
            NextX:=CurrentX+(StepDir*StepSize);
            TPWrite "Pass2: NextX=" \Num:=NextX;

            ! Check if pass complete (no more columns to step to)
            IF (StepDir=1 AND NextX>WorkMaxX) OR (StepDir=-1 AND NextX<WorkMinX) THEN
                TPWrite "Pass2: EXIT - NextX out of bounds";
                FCPressEnd Offs(pHeliEnd,0,0,50),v100,\DeactOnly,tHeli\WObj:=Bed1Wyong;
                EXIT;
            ENDIF

            ! Clamp to bounds
            IF NextX>WorkMaxX THEN
                NextX:=WorkMaxX;
            ELSEIF NextX<WorkMinX THEN
                NextX:=WorkMinX;
            ENDIF

            ! Step to next X column
            TPWrite "Pass2: Step to X=" \Num:=NextX;
            pHeliEnd.trans.x:=-NextX;
            pHeliEnd.extax.eax_a:=Bed1Wyong.uframe.trans.x-NextX;
            FCPressL pHeliEnd,vHeliTravel,CurrentForce,fine,tHeli\WObj:=Bed1Wyong;
            CurrentX:=NextX;

            ! Flip sweep direction for next Y sweep
            SweepDir:=-SweepDir;
            IF SweepDir=1 THEN
                EndY:=WorkMinY;
            ELSE
                EndY:=WorkMaxY;
            ENDIF

            ! Set up end position and sweep Y
            TPWrite "Pass2: Sweep Y to " \Num:=EndY;
            pHeliEnd.trans.y:=EndY;
            FCPressL pHeliEnd,vHeliTravel,CurrentForce,fine,tHeli\WObj:=Bed1Wyong;
        ENDWHILE
        TPWrite "=== PASS 2 COMPLETE ===";

        ! === LIFT OFF BED ===
        pHeliPos.trans.z:=SafeZ;
        MoveL pHeliPos,v100,z5,tHeli\WObj:=Bed1Wyong;

        ! === STOP BLADE ROTATION ===
        HeliBladeSpeed 0,"FWD";
        WaitTime\InPos,3;

        ConfL\On;
        ConfJ\On;

        ! === PACKAWAY ===
        Heli_Dropoff;
        Home;

        TPWrite "PyHeli Complete";
    ERROR
        HeliBladeSpeed 0,"FWD";
        RAISE;
    ENDPROC


    PROC PyVac()
        ! PyVac - Vacuum procedure with serpentine pattern
        ! Workzone: bed
        ! Generated by Onyx Toolpath Generator

        VAR robtarget pVacPos;
        VAR robtarget pVacEnd;
        VAR num VacZ:=-20;
        VAR num SafeZ:=300;

        ! Force control parameters
        VAR num VacForce:=50;
        VAR num VacZMin:=-20;
        VAR num VacZMax:=50;
        VAR num VacZRange:=70;

        ! Workspace bounds (with offsets applied)
        VAR num WorkMinX:=0;
        VAR num WorkMaxX:=8500;
        VAR num WorkMinY:=0;
        VAR num WorkMaxY:=1650;

        ! Pattern parameters
        VAR num StepSize:=300;
        VAR num SweepDir:=-1;
        VAR num YStepDir:=-1;
        VAR num CurrentY:=1650;
        VAR num NextY;
        VAR num StartX;
        VAR num EndX;

        VAR speeddata vVac:=[200,30,2000,15];
        VAR num NumPasses;

        NumPasses:=Trunc(Abs(WorkMaxY-WorkMinY)/StepSize)+1;

        TPWrite "PyVac: Serpentine Pattern";
        TPWrite "Work Area (8500,1650) to (0,0)";
        TPWrite "Passes=" \Num:=NumPasses;
        TPWrite "Step=" \Num:=StepSize;
        TPWrite "Speed=" \Num:=200;

        IF ToolNum<>5 THEN
            TPWrite "PyVac: ToolNum<>5, need pickup";
            TPWrite "PyVac: ToolNum=" \Num:=ToolNum;
            TPWrite "PyVac: Calling Vac_Pickup...";
            Stop;
            Vac_Pickup;
            TPWrite "PyVac: Vac_Pickup complete";
        ELSE
            CurrentJoints:=CJointT();
            CurrentPos:=CalcRobT(CurrentJoints,tVac\WObj:=Bed1Wyong);
            IF CurrentPos.trans.z<SafeZ THEN
                MoveL Offs(CurrentPos,0,0,(SafeZ-CurrentPos.trans.z)),v500,z5,tVac\WObj:=Bed1Wyong;
            ENDIF
        ENDIF

        ConfL\Off;
        ConfJ\Off;

        pVacPos:=[[0,0,VacZ],[0.00615322,-0.709926,0.704246,-0.00239206],[1,-1,0,0],[0,9E+09,9E+09,9E+09,9E+09,9E+09]];

        TPWrite "Press Play to start";
        Stop;

        Vac_on;

        ! Main vacuum loop - always sweep right to left, lift and return
        WHILE TRUE DO
            ! Move to row start above work surface (right side)
            pVacPos.trans.x:=-WorkMaxX;
            pVacPos.trans.y:=CurrentY;
            pVacPos.trans.z:=VacZMax;
            pVacPos.extax.eax_a:=Bed1Wyong.uframe.trans.x-WorkMaxX;
            MoveL pVacPos,vVac,fine,tVac\WObj:=Bed1Wyong;

            ! Set up end position
            pVacEnd:=pVacPos;
            pVacEnd.trans.x:=-WorkMinX;
            pVacEnd.trans.z:=VacZ;
            pVacEnd.extax.eax_a:=Bed1Wyong.uframe.trans.x-WorkMinX;

            ! Sweep right to left
            pVacPos.trans.z:=VacZ;
            MoveL pVacPos,vVac,fine,tVac\WObj:=Bed1Wyong;
            MoveL pVacEnd,vVac,z5,tVac\WObj:=Bed1Wyong;

            ! Calculate next row
            NextY:=CurrentY+(YStepDir*StepSize);

            ! Check if pattern complete
            IF (YStepDir=1 AND NextY>WorkMaxY) OR (YStepDir=-1 AND NextY<WorkMinY) THEN
                ! Pattern complete
                EXIT;
            ENDIF

            ! Clamp to bounds for partial last step
            IF NextY>WorkMaxY THEN
                NextY:=WorkMaxY;
            ELSEIF NextY<WorkMinY THEN
                NextY:=WorkMinY;
            ENDIF

            ! Lift off work surface (already lifted by FCPressEnd)
            pVacPos.trans.z:=SafeZ;
            pVacPos.trans.x:=-WorkMinX;
            pVacPos.extax.eax_a:=Bed1Wyong.uframe.trans.x-WorkMinX;
            MoveL pVacPos,v500,z5,tVac\WObj:=Bed1Wyong;

            ! Return to start X (right side) at safe height, step to next Y
            pVacPos.trans.x:=-WorkMaxX;
            pVacPos.trans.y:=NextY;
            pVacPos.extax.eax_a:=Bed1Wyong.uframe.trans.x-WorkMaxX;
            MoveL pVacPos,v500,z5,tVac\WObj:=Bed1Wyong;

            CurrentY:=NextY;
        ENDWHILE

        Vac_off;

        pVacPos.trans.z:=SafeZ;
        MoveL pVacPos,v100,z5,tVac\WObj:=Bed1Wyong;

        ConfL\On;
        ConfJ\On;

        Vac_Dropoff;
        Home;

        TPWrite "PyVac Complete";
    ERROR
        Vac_off;
        RAISE;
    ENDPROC


    PROC PyPolish()
        ! PyPolish - Polisher serpentine with force control
        ! Workzone: bed
        ! Generated by Onyx Toolpath Generator

        VAR robtarget pPolPos;
        VAR robtarget pPolEnd;
        VAR num PolZ:=0;
        VAR num SafeZ:=300;

        ! Force control parameters
        VAR num StartForce:=300;
        VAR num MotionForce:=300;
        VAR num ForceChange:=100;
        VAR num PosSupvDist:=100;

        ! Workspace bounds (with offsets applied)
        VAR num WorkMinX:=0;
        VAR num WorkMaxX:=8500;
        VAR num WorkMinY:=0;
        VAR num WorkMaxY:=1650;

        ! Pattern parameters
        VAR num StepSize:=300;
        VAR num SweepDir:=1;
        VAR num YStepDir:=-1;
        VAR num CurrentY:=1650;
        VAR num NextY;
        VAR num StartX;
        VAR num EndX;

        VAR speeddata vPolApproach:=[20,30,2000,15];
        VAR speeddata vPolRetract:=[50,30,2000,15];
        VAR speeddata vPolTravel:=[100,30,2000,15];
        VAR num NumPasses;

        NumPasses:=Trunc(Abs(WorkMaxY-WorkMinY)/StepSize)+1;

        TPWrite "PyPolish: Serpentine Pattern";
        TPWrite "Work Area (8500,1650) to (0,0)";
        TPWrite "Passes=" \Num:=NumPasses;
        TPWrite "Step=" \Num:=StepSize;
        TPWrite "Force=" \Num:=MotionForce;

        IF ToolNum<>6 THEN
            TPWrite "PyPolish: ToolNum<>6, need pickup";
            Stop;
            Home;
            Polish_Pickup;
        ELSE
            CurrentJoints:=CJointT();
            CurrentPos:=CalcRobT(CurrentJoints,tPolish\WObj:=Bed1Wyong);
            IF CurrentPos.trans.z<SafeZ THEN
                MoveL Offs(CurrentPos,0,0,(SafeZ-CurrentPos.trans.z)),v500,z5,tPolish\WObj:=Bed1Wyong;
            ENDIF
        ENDIF

        ConfL\Off;
        ConfJ\Off;

        ! Set start/end based on sweep direction
        IF SweepDir=1 THEN
            StartX:=WorkMinX;
            EndX:=WorkMaxX;
        ELSE
            StartX:=WorkMaxX;
            EndX:=WorkMinX;
        ENDIF

        ! Set initial position with fixed orientation (facing +X direction)
        pPolPos:=[[0,0,PolZ],OrientZYX(0,0,180),[1,-1,-1,0],[0,9E+09,9E+09,9E+09,9E+09,9E+09]];

        ! Calibrate force control
        FCCalib PolishLoad;

        TPWrite "Press Play to start";
        Stop;

        ! Move to row start above surface
        pPolPos.trans.x:=-StartX;
        pPolPos.trans.y:=CurrentY;
        pPolPos.trans.z:=SafeZ;
        pPolPos.extax.eax_a:=Bed1Wyong.uframe.trans.x-StartX;
        MoveL pPolPos,vPolTravel,z5,tPolish\WObj:=Bed1Wyong;

        ! Lower to approach height
        pPolPos.trans.z:=PolZ+50;
        MoveL pPolPos,vPolApproach,fine,tPolish\WObj:=Bed1Wyong;

        ! Turn on polisher and wait for spin-up
        Pol_off;
        WaitTime 0.2;
        Pol_on;
        WaitTime 1.0;

        ! Set up end position for first sweep
        pPolEnd:=pPolPos;
        pPolEnd.trans.x:=-EndX;
        pPolEnd.trans.z:=PolZ;
        pPolEnd.extax.eax_a:=Bed1Wyong.uframe.trans.x-EndX;

        ! Start force control
        FCPress1LStart Offs(pPolPos,0,0,25),vPolApproach,\Fz:=StartForce,15,\ForceChange:=ForceChange\PosSupvDist:=PosSupvDist,z5,tPolish\WObj:=Bed1Wyong;

        ! Main polisher loop - stays in contact during serpentine
        WHILE TRUE DO
            ! === SWEEP X (full length) ===
            FCPressL pPolEnd,vPolTravel,MotionForce,fine,tPolish\WObj:=Bed1Wyong;

            ! Calculate next row
            NextY:=CurrentY+(YStepDir*StepSize);

            ! Check if pattern complete
            IF (YStepDir=1 AND NextY>WorkMaxY) OR (YStepDir=-1 AND NextY<WorkMinY) THEN
                FCPressEnd Offs(pPolEnd,0,0,50),vPolRetract,\DeactOnly,tPolish\WObj:=Bed1Wyong;
                Pol_off;
                EXIT;
            ENDIF

            ! Clamp to bounds
            IF NextY>WorkMaxY THEN
                NextY:=WorkMaxY;
            ELSEIF NextY<WorkMinY THEN
                NextY:=WorkMinY;
            ENDIF

            ! Step to next Y row (still in force control)
            pPolEnd.trans.y:=NextY;
            FCPressL pPolEnd,vPolTravel,MotionForce,fine,tPolish\WObj:=Bed1Wyong;
            CurrentY:=NextY;

            ! Flip sweep direction
            SweepDir:=-SweepDir;
            IF SweepDir=1 THEN
                StartX:=WorkMinX;
                EndX:=WorkMaxX;
            ELSE
                StartX:=WorkMaxX;
                EndX:=WorkMinX;
            ENDIF

            ! Set up end position for next sweep
            pPolEnd.trans.x:=-EndX;
            pPolEnd.extax.eax_a:=Bed1Wyong.uframe.trans.x-EndX;
        ENDWHILE

        ! Return to safe height
        pPolPos.trans.z:=SafeZ;
        MoveL pPolPos,vPolTravel,z5,tPolish\WObj:=Bed1Wyong;

        ConfL\On;
        ConfJ\On;

        Polish_Dropoff;
        Home;

        TPWrite "PyPolish Complete";
    ERROR
        Pol_off;
        RAISE;
    ENDPROC


    PROC PyVibScreed()
        ! PyVibScreed - Vibrating Screed with Panel workzone parameters
        ! Workzone: Panel
        ! Panel: X=1900 to 6550, Y=700, Z=150
        ! Panel Start/Finish Offset: 200 mm
        ! Actual travel: X=1700 to 6750
        ! Global Z Offset: 0 mm
        ! Screed Z Offset: 4 mm
        ! Working Z: 154 mm
        ! Speed: 50 mm/s
        ! Angle: 11°
        ! Generated by Onyx Toolpath Generator

        VAR robtarget pScreedPos;
        VAR robtarget pScreedEnd;
        VAR num ScrStartX:=1700;
        VAR num ScrEndX:=6750;
        VAR num ScrY:=700;
        VAR num WorkZ:=154;
        VAR num SafeZ:=500;
        VAR num ScrAoffset:=11;
        VAR speeddata vScreed:=[50,30,2000,15];

        TPWrite "PyVibScreed: Panel Workzone";
        TPWrite "Start X=" \Num:=ScrStartX;
        TPWrite "End X=" \Num:=ScrEndX;
        TPWrite "Y=" \Num:=ScrY;
        TPWrite "Work Z=" \Num:=WorkZ;
        TPWrite "Speed=" \Num:=50;
        TPWrite "Angle=" \Num:=ScrAoffset;

        CurrentJoints:=CJointT();
        CurrentPos:=CalcRobT(CurrentJoints,tVS\WObj:=Bed1Wyong);

        IF ToolNum<>3 THEN
            TPWrite "PyVibScreed: ToolNum<>3, need pickup";
            Stop;
            Home;
            VS_Pickup;
        ELSEIF (CurrentPos.trans.z<SafeZ) THEN
            MoveL Offs(CurrentPos,0,0,(SafeZ-CurrentPos.trans.z)),v200,z5,tVS\WObj:=Bed1Wyong;
        ENDIF

        ! Set up start position - use pVSstart as template for rotation
        pScreedPos:=pVSstart;
        pScreedPos.trans.x:=-ScrStartX;
        pScreedPos.trans.y:=ScrY;
        pScreedPos.trans.z:=SafeZ;
        pScreedPos.extax.eax_a:=Bed1Wyong.uframe.trans.x-ScrStartX+700;

        ! Set up end position
        pScreedEnd:=pScreedPos;
        pScreedEnd.trans.x:=-ScrEndX;
        pScreedEnd.trans.z:=WorkZ;
        pScreedEnd.extax.eax_a:=Bed1Wyong.uframe.trans.x-ScrEndX+700;

        ! Move to start position at safe height (holding high)
        MoveL pScreedPos,v500,fine,tVS\WObj:=Bed1Wyong;

        ! Drop down to approach height (100mm above work)
        pScreedPos.trans.z:=WorkZ+100;
        MoveL RelTool(pScreedPos,0,0,0\Ry:=ScrAoffset),v200,fine,tVS\WObj:=Bed1Wyong;

        ! Start vibrator
        VS_on;

        ! Lower to working Z
        pScreedPos.trans.z:=WorkZ;
        MoveL RelTool(pScreedPos,0,0,0\Ry:=ScrAoffset),v50,z5,tVS\WObj:=Bed1Wyong;

        ! Screed across panel
        MoveL RelTool(pScreedEnd,0,0,0\Ry:=ScrAoffset),vScreed,z5,tVS\WObj:=Bed1Wyong;

        ! Lift off at end
        pScreedEnd.trans.z:=WorkZ+100;
        MoveL RelTool(pScreedEnd,0,0,0\Ry:=ScrAoffset),v100,z5,tVS\WObj:=Bed1Wyong;

        VS_off;

        ! Return to safe height
        pScreedEnd.trans.z:=SafeZ;
        MoveL pScreedEnd,v200,z5,tVS\WObj:=Bed1Wyong;

        VS_Dropoff;

        TPWrite "PyVibScreed Complete";
    ENDPROC


    PROC PyPan()
        ! Python-generated Pan procedure
        ! Serpentine pattern over Panel workzone

        VAR robtarget pPanPos;
        VAR robtarget pPanEnd;
        VAR robtarget CurrentPos;
        VAR jointtarget CurrentJoints;

        ! Workspace bounds (Panel)
        CONST num WorkMinX:=1900;
        CONST num WorkMaxX:=6550;
        CONST num WorkMinY:=700;
        CONST num WorkMaxY:=2100;
        CONST num PanZ:=151;
        CONST num SafeZ:=451;

        ! Pattern parameters
        VAR num StepSize:=500;
        VAR num SweepDir:=1;
        VAR num StepDir:=-1;
        VAR num CurrentY:=2100;
        VAR num CurrentX:=1900;
        VAR num NextY;
        VAR num NextX;
        VAR num StartX;
        VAR num EndX;
        VAR num StartY;
        VAR num EndY;

        ! Speed and blade parameters
        VAR num PanSpeed:=140;
        VAR num PanAngle:=0;  ! Pan always uses 0 blade angle
        VAR speeddata vPanTravel:=[500,30,2000,15];
        VAR num NumPasses;

        NumPasses:=Trunc(Abs(WorkMaxY-WorkMinY)/StepSize)+1;

        TPWrite "PyPan: Serpentine Pattern";
        TPWrite "Work Area (6550,2100) to (1900,700)";
        TPWrite "Passes=" \Num:=NumPasses;
        TPWrite "Step=" \Num:=StepSize;

        IF ToolNum<>2 THEN
            TPWrite "PyPan: ToolNum<>2, need pickup";
            Stop;
            Home;
            Heli_Pickup;
        ELSE
            CurrentJoints:=CJointT();
            CurrentPos:=CalcRobT(CurrentJoints,tHeli\WObj:=Bed1Wyong);
            IF CurrentPos.trans.z<SafeZ THEN
                MoveL Offs(CurrentPos,0,0,(SafeZ-CurrentPos.trans.z)),v500,z5,tHeli\WObj:=Bed1Wyong;
            ENDIF
        ENDIF

        ! Set start/end based on sweep direction
        IF SweepDir=1 THEN
            StartX:=WorkMinX;
            EndX:=WorkMaxX;
        ELSE
            StartX:=WorkMaxX;
            EndX:=WorkMinX;
        ENDIF

        ! Set initial position with fixed orientation
        pPanPos:=[[0,0,PanZ],OrientZYX(0,0,180),[0,0,0,0],[0,9E+09,9E+09,9E+09,9E+09,9E+09]];

        ! Move to row start above surface
        pPanPos.trans.x:=-StartX;
        pPanPos.trans.y:=CurrentY;
        pPanPos.trans.z:=SafeZ;
        pPanPos.extax.eax_a:=Bed1Wyong.uframe.trans.x-StartX;
        MoveJ pPanPos,v500,z5,tHeli\WObj:=Bed1Wyong;

        TPWrite "Press Play to start";
        Stop;

        ! Disable configuration tracking for serpentine movements
        ConfL\Off;
        ConfJ\Off;

        ! Lower to working height
        pPanPos.trans.z:=PanZ;
        MoveL pPanPos,v50,fine,tHeli\WObj:=Bed1Wyong;

        ! Start blade rotation
        HeliBladeSpeed PanSpeed,"FWD";
        WaitTime\InPos,3;

        ! Set up end position for first sweep
        pPanEnd:=pPanPos;
        pPanEnd.trans.x:=-EndX;
        pPanEnd.extax.eax_a:=Bed1Wyong.uframe.trans.x-EndX;

        ! ========== PASS 1: X-direction sweeps (stepping in Y) ===========
        WHILE TRUE DO
            ! === SWEEP X (full length) ===
            MoveL pPanEnd,vPanTravel,z5,tHeli\WObj:=Bed1Wyong;

            ! Calculate next row
            NextY:=CurrentY+(StepDir*StepSize);

            ! Check if pass complete
            IF (StepDir=1 AND NextY>WorkMaxY) OR (StepDir=-1 AND NextY<WorkMinY) THEN
                EXIT;
            ENDIF

            ! Clamp to bounds
            IF NextY>WorkMaxY THEN
                NextY:=WorkMaxY;
            ELSEIF NextY<WorkMinY THEN
                NextY:=WorkMinY;
            ENDIF

            ! Step to next Y row
            pPanEnd.trans.y:=NextY;
            MoveL pPanEnd,vPanTravel,z5,tHeli\WObj:=Bed1Wyong;
            CurrentY:=NextY;

            ! Flip sweep direction
            SweepDir:=-SweepDir;
            IF SweepDir=1 THEN
                StartX:=WorkMinX;
                EndX:=WorkMaxX;
            ELSE
                StartX:=WorkMaxX;
                EndX:=WorkMinX;
            ENDIF

            ! Set up end position for next sweep
            pPanEnd.trans.x:=-EndX;
            pPanEnd.extax.eax_a:=Bed1Wyong.uframe.trans.x-EndX;
        ENDWHILE

        ! ========== PASS 2: Y-direction sweeps (stepping in X) ==========

        ! Reset for Y-direction passes - start from current position
        CurrentX:=Abs(pPanEnd.trans.x);

        ! Determine step direction based on where Pass 1 ended
        ! At high X, step toward low X; at low X, step toward high X
        IF CurrentX>((WorkMinX+WorkMaxX)/2) THEN
            StepDir:=-1;
        ELSE
            StepDir:=1;
        ENDIF

        SweepDir:=1;
        StartY:=WorkMaxY;
        EndY:=WorkMinY;

        ! Set up for Y sweep and move to start position
        pPanEnd.trans.y:=EndY;
        MoveL pPanEnd,vPanTravel,z5,tHeli\WObj:=Bed1Wyong;

        WHILE TRUE DO
            ! Calculate next column
            NextX:=CurrentX+(StepDir*StepSize);

            ! Check if pass complete
            IF (StepDir=1 AND NextX>WorkMaxX) OR (StepDir=-1 AND NextX<WorkMinX) THEN
                EXIT;
            ENDIF

            ! Clamp to bounds
            IF NextX>WorkMaxX THEN
                NextX:=WorkMaxX;
            ELSEIF NextX<WorkMinX THEN
                NextX:=WorkMinX;
            ENDIF

            ! Step to next X column
            pPanEnd.trans.x:=-NextX;
            pPanEnd.extax.eax_a:=Bed1Wyong.uframe.trans.x-NextX;
            MoveL pPanEnd,vPanTravel,z5,tHeli\WObj:=Bed1Wyong;
            CurrentX:=NextX;

            ! Flip sweep direction
            SweepDir:=-SweepDir;
            IF SweepDir=1 THEN
                StartY:=WorkMinY;
                EndY:=WorkMaxY;
            ELSE
                StartY:=WorkMaxY;
                EndY:=WorkMinY;
            ENDIF

            ! Set up end position for next sweep
            pPanEnd.trans.y:=EndY;

            ! === SWEEP Y (full length) ===
            MoveL pPanEnd,vPanTravel,z5,tHeli\WObj:=Bed1Wyong;
        ENDWHILE

        ! === LIFT OFF BED ===
        pPanPos.trans.z:=SafeZ;
        MoveL pPanPos,v100,z5,tHeli\WObj:=Bed1Wyong;

        ! === STOP BLADE ROTATION ===
        HeliBladeSpeed 0,"FWD";
        WaitTime\InPos,3;

        ConfL\On;
        ConfJ\On;

        ! === PACKAWAY ===
        Heli_Dropoff;
        Home;

        TPWrite "PyPan Complete";
    ENDPROC

ENDMODULE
